(* Logix 5000 project; controller Prueba2 vendor 1 type 14 code 156 rev 30.11; software revision 30.00 *)

TASK MainTask (continuous, watchdog 500 ms) : MainProgram

MODULES
   Local : vendor 1 type 14 code 156 (Compact 0, rev 30.11)
      DI_4 : 1769-IQ16 (Compact 4, rev 1.1, Input RPI 20 ms)
      DO_5 : vendor 1 type 7 code 86 (Compact 5, rev 2.1, Output RPI 20 ms)
END_MODULES

VAR_GLOBAL   (* controller tags *)
   Count_S1 : COUNTER := (PRE := 3);
   GD_IN_0 : BOOL;
   GD_IN_1 : BOOL;
   GD_IN_2 : BOOL;   // GD sensor 1
   GD_IN_3 : BOOL := 1;
   GD_IN_4 : BOOL;
   GD_IN_5 : BOOL;   // GD RESET
   GD_OUT_0 : BOOL;
   GD_OUT_1 : BOOL;
   SENSOR : BOOL;
   TagA : BOOL;
   TIMER1 : TIMER := (PRE := 5000);
END_VAR

PROGRAM MainProgram   (* main routine MainRoutine *)
VAR
   PS_BANDA1 : ALIAS FOR Local:5:O.Data.0;
   PS_START : ALIAS FOR Local:4:I.Data.1;
   PS_STOP : ALIAS FOR Local:4:I.Data.0;
END_VAR

ROUTINE MainRoutine   (* ladder *)
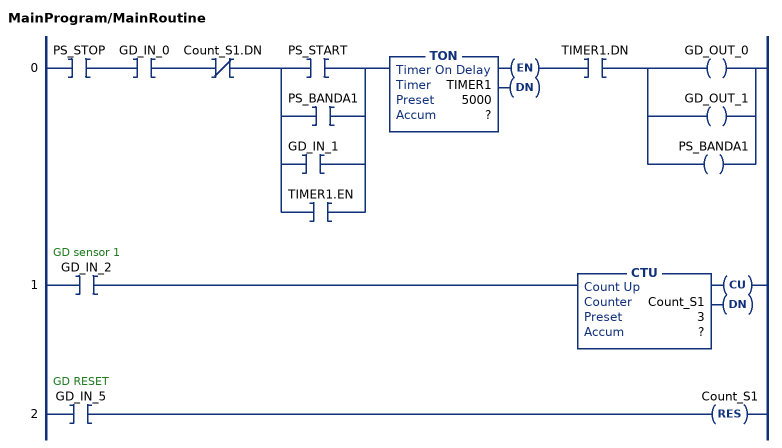
   0: XIC(PS_STOP)XIC(GD_IN_0)XIO(Count_S1.DN)[XIC(PS_START) ,[XIC(PS_BANDA1) ,[XIC(GD_IN_1) ,XIC(TIMER1.EN) ] ] ]TON(TIMER1,?,?)XIC(TIMER1.DN)[OTE(GD_OUT_0) ,[OTE(GD_OUT_1) ,OTE(PS_BANDA1) ] ];
   1: XIC(GD_IN_2)CTU(Count_S1,?,?);
   2: XIC(GD_IN_5)RES(Count_S1);
END_ROUTINE
END_PROGRAM
